FUNCTION_BLOCK CylinderMech
VAR_INPUT
	//PressureBoreSide : LREAL;
	//PressureRodSide : LREAL;
	param : ST_pValveControlledCylinder;
	F_Hydraulic : LREAL;
END_VAR
VAR_OUTPUT
	PistonAcceleration: LREAL;
	PistonVelocity : LREAL;
	PistonPosition : LREAL;
	F_Piston : LREAL;
END_VAR
VAR
	ssMethodType : SINT := 1; 
	fbPistonVelocity : DiscreteTimeIntegrator_Init;
	fbPistonPosition : DiscreteTimeIntegrator_Init;
	y_tmp : LREAL;
	SpringContactCoefficient : LREAL;
	DamperContactCoefficient : LREAL;
	F_Upper_Stroke_Limit : LREAL;
	F_Lower_Stroke_Limit : LREAL;
	F_Stribeck_Friction : LREAL;
	AbsPosition: LREAL;
END_VAR

// Upper Stroke Limit Contact Force [N] //
IF PistonPosition >= param.xMax THEN 
	SpringContactCoefficient := param.cyl_k_end;
ELSIF PistonPosition < param.xMax THEN 
	SpringContactCoefficient := 0;
END_IF;	

IF PistonPosition >= param.xMax THEN 
	DamperContactCoefficient := param.cyl_c_end;
ELSIF PistonPosition < param.xMax THEN 
	DamperContactCoefficient := 0;
END_IF;	

F_Upper_Stroke_Limit := ((PistonPosition - param.xMax) * SpringContactCoefficient) + (DamperContactCoefficient * PistonVelocity);



//// Lower Stroke Limit Contact Force [N] //
IF PistonPosition > 0 THEN 
	SpringContactCoefficient := 0;
ELSIF PistonPosition <= 0 THEN 
	SpringContactCoefficient := param.cyl_k_end;
END_IF;	

IF PistonPosition > 0 THEN 
	DamperContactCoefficient := 0;
ELSIF PistonPosition <= 0 THEN 
	DamperContactCoefficient := param.cyl_c_end;
END_IF;	

AbsPosition := ABS(PistonPosition);
F_Lower_Stroke_Limit := (SpringContactCoefficient * AbsPosition) + (DamperContactCoefficient * (-1) * PistonVelocity);



//// Stribeck Friction Force [N] //
//y_tmp := EXP((PistonVelocity * param.FrictionForceApproximationConstant) * 2.0);
//y_tmp := (y_tmp - 1.0) / (y_tmp + 1.0);
//F_Stribeck_Friction := (((EXP(( -(PistonVelocity * y_tmp)) / param.StaticFrictionTimeConstant) * ABS(param.StaticFrictionForce)) + param.ColoumbFriction) * y_tmp) + (PistonVelocity * param.ViscousFrictionCoefficient);


/// Piston Force Total [N] ///
F_Piston := ( (F_Hydraulic - F_Upper_Stroke_Limit + F_Lower_Stroke_Limit - F_Stribeck_Friction) ) * 4;


// Piston Acceleration [m/s^2]
PistonAcceleration := (F_Piston - param.ExternalForce) / param.EffectiveMass;

PistonVelocity := Work.VpistonMainBoom; 	//From Unreal engine
PistonPosition := Work.XpistonMainBoom;		//From Unreal engine

//fbPistonVelocity(
//	ssMethodType := ssMethodType,
//	tCycle := param.tCycle,
//	In := PistonAcceleration,
//	Init := param.v0,
//	minOut := -param.vMax,
//	maxOut := param.vMax,
//	Out => PistonVelocity
//	);

//fbPistonPosition(
//	ssMethodType := ssMethodType,
//	tCycle := param.tCycle,
//	In := PistonVelocity,
//	Init := param.x0,
//	minOut := -5000,
//	maxOut := param.xMax+5000,
//	Out => PistonPosition
//	);

//IF PistonPosition >= param.xMax THEN 
//	PistonPosition := param.xMax;
//ELSIF PistonPosition <= 0 THEN 
//	PistonPosition := 0;
//END_IF;

END_FUNCTION_BLOCK

(* stored: Version 1.1.0.1, ProductVersion 3.1.4024.9
   POU CylinderMech: Id {3bf06456-7c7d-48f2-a9cc-e4b64f4dae07}, SpecialFunc None *)
